{attribute addProperty BoxType "EK1122-0000-0018"}
{attribute addProperty Id "Beckhoff_EQ3xxxsub_EK1100EK1100_179A0949162A_0001_EQ3174_0002_0016EQ3174_6082EBFD21026.25A_0002_EQ3174_0002_0017EQ3174_6082EBFD21026.25A_0003_EQ3174_0002_0021EQ3174_6082EBFD21026.25A_0004_EQ3174_0002_0022EQ3174_B7B5302521026.25A_0005_EQ3174_0002_0023EQ3174_B7B5302521026.25A_0006_EQ3204_0002_0016EQ3204_72ABB95437847.25A_0007_EQ3204_0002_0017EQ3204_72ABB95437847.25A_0008_EQ3204_0002_0020EQ3204_72ABB95437847.25A_0009_EQ3204_0002_0021EQ3204_C91659E221026.25A_0010_EQ3204_0002_0022EQ3204_C91659E221026.25A_0011_EQ3314_0002_0016EQ3314_1D3C92AC21026.25A_0012_EQ3314_0002_0017EQ3314_1D3C92AC21026.25A_0013_EQ3314_0002_0021EQ3314_1D3C92AC21026.25A_0014_EQ3314_0002_0022EQ3314_A69716D721026.25"}
{attribute addProperty CRC "3266874225"}
{attribute addProperty SizeInBites "3460"}
{attribute addProperty SizeInBytes "432.5"}
TYPE Beckhoff_EQ3xxxEK1122_C2B88B71 EXTENDS EK1122_179A0949 :
STRUCT
	{attribute addProperty Name "Beckhoff_EQ3xxxsub_EK1100"}
	Beckhoff_EQ3xxxsub_EK1100 : EK1100_179A0949;
	{attribute addProperty Name "A_0001_EQ3174_0002_0016"}
	A_0001_EQ3174_0002_0016 : EQ3174_6082EBFD;
	{attribute addProperty Name "A_0002_EQ3174_0002_0017"}
	A_0002_EQ3174_0002_0017 : EQ3174_6082EBFD;
	{attribute addProperty Name "A_0003_EQ3174_0002_0021"}
	A_0003_EQ3174_0002_0021 : EQ3174_6082EBFD;
	{attribute addProperty Name "A_0004_EQ3174_0002_0022"}
	A_0004_EQ3174_0002_0022 : EQ3174_B7B53025;
	{attribute addProperty Name "A_0005_EQ3174_0002_0023"}
	A_0005_EQ3174_0002_0023 : EQ3174_B7B53025;
	{attribute addProperty Name "A_0006_EQ3204_0002_0016"}
	A_0006_EQ3204_0002_0016 : EQ3204_72ABB954;
	{attribute addProperty Name "A_0007_EQ3204_0002_0017"}
	A_0007_EQ3204_0002_0017 : EQ3204_72ABB954;
	{attribute addProperty Name "A_0008_EQ3204_0002_0020"}
	A_0008_EQ3204_0002_0020 : EQ3204_72ABB954;
	{attribute addProperty Name "A_0009_EQ3204_0002_0021"}
	A_0009_EQ3204_0002_0021 : EQ3204_C91659E2;
	{attribute addProperty Name "A_0010_EQ3204_0002_0022"}
	A_0010_EQ3204_0002_0022 : EQ3204_C91659E2;
	{attribute addProperty Name "A_0011_EQ3314_0002_0016"}
	A_0011_EQ3314_0002_0016 : EQ3314_1D3C92AC;
	{attribute addProperty Name "A_0012_EQ3314_0002_0017"}
	A_0012_EQ3314_0002_0017 : EQ3314_1D3C92AC;
	{attribute addProperty Name "A_0013_EQ3314_0002_0021"}
	A_0013_EQ3314_0002_0021 : EQ3314_1D3C92AC;
	{attribute addProperty Name "A_0014_EQ3314_0002_0022"}
	A_0014_EQ3314_0002_0022 : EQ3314_A69716D7;
END_STRUCT
END_TYPE

(* stored: Version 1.2.0.0, ProductVersion 3.1.4024.9
   DUT Beckhoff_EQ3xxxEK1122_C2B88B71: Id {6cd1296b-fb59-47f8-b48a-a8b415237374} *)
